# EPICS autosave request: ipApp/Db/caen_N8031_settings.req
$(P)$(R)CH0:Name.VAL
$(P)$(R)CH1:Name.VAL
$(P)$(R)CH2:Name.VAL
$(P)$(R)CH3:Name.VAL
$(P)$(R)CH4:Name.VAL
$(P)$(R)CH5:Name.VAL
$(P)$(R)CH6:Name.VAL
$(P)$(R)CH7:Name.VAL
